//Placeholder, WIP --> need to define what purpose this struct serves
TYPE ST_SubSystem :
STRUCT
    refIn: REFERENCE TO ST_SubSystemIn;
    refOut: REFERENCE TO ST_SubSystemOut;
END_STRUCT
END_TYPE

(* stored: Version 1.1.0.1
   DUT ST_SubSystem: Id {389ba33d-0a84-02f2-3a99-f7b12e821d76} *)
